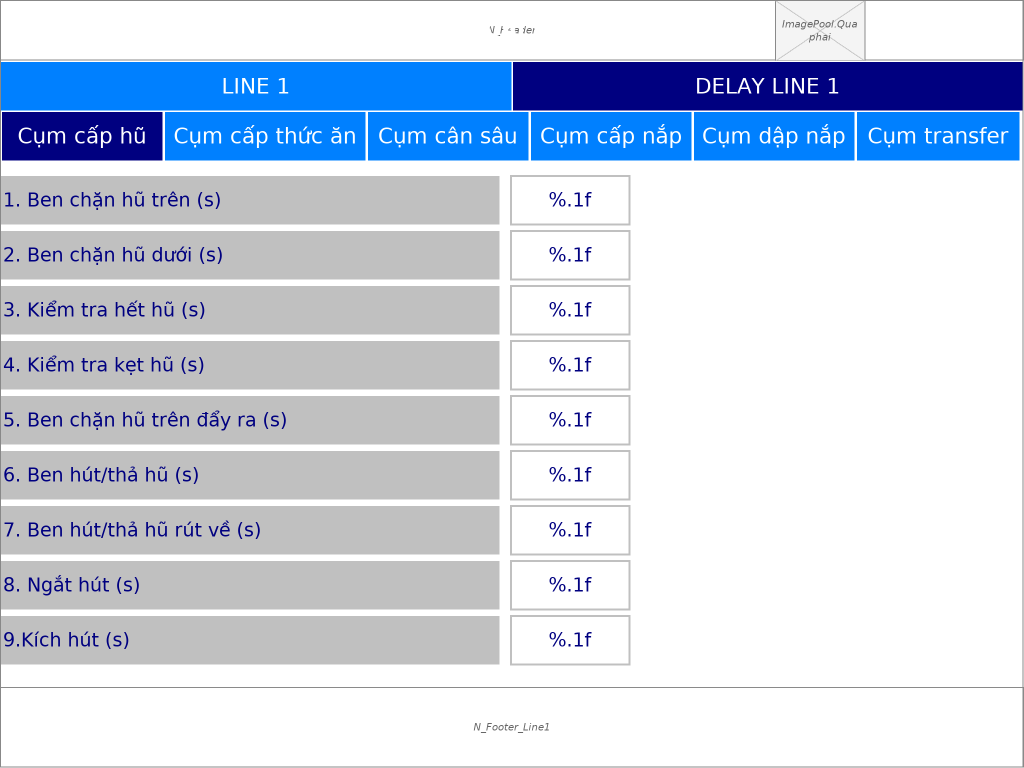
VISUALIZATION N_Setting_Delay_JarSupply1  // 1024x768
    Frame (0,687 1024x80)
        shows N_Footer_Line1()
    Frame (0,0 1024x60)
        shows N_Header()
    Textfield (353,4 420x50), "MÀN HÌNH CÀI KHOẢNG TRỄ LINE 1"
    Rectangle (0,61 512x50), "LINE 1"
        OnMouseClick: change screen: N_Setting_Line1
    Image (775,0 90x61), image: ImagePool.Qua phai
        OnMouseClick: change screen: N_Setting_Delay_JarSupply2
    Rectangle (1,111 162x50), "Cụm cấp hũ"
        OnMouseClick: change screen: N_Setting_Delay_JarSupply1
    Rectangle (164,111 202x50), "Cụm cấp thức ăn"
        OnMouseClick: change screen: N_Setting_Delay_FoodSupply1
    Rectangle (367,111 162x50), "Cụm cân sâu"
        OnMouseClick: change screen: N_Setting_Delay_WormWeight1
    Rectangle (530,111 162x50), "Cụm cấp nắp"
        OnMouseClick: change screen: N_Setting_Delay_LidSupply1
    Rectangle (693,111 162x50), "Cụm dập nắp"
        OnMouseClick: change screen: N_Setting_Delay_LidPressing1
    Rectangle (856,111 164x50), "Cụm transfer"
        OnMouseClick: change screen: N_Setting_Delay_Tranfer1
    Rectangle (512,61 511x50), "DELAY LINE 1"
        OnMouseClick: change screen: N_Setting_Delay_JarSupply1
    Rectangle (0,175 500x50), "1. Ben chặn hũ trên (s)"
    Rectangle (510,175 120x50), "%.1f", text variable: PR_Line01.timerCheckCylinder_Up
        OnMouseClick: write PR_Line01.timerCheckCylinder_Up via VisuDialogs.Numpad
    Rectangle (0,230 500x50), "2. Ben chặn hũ dưới (s)"
    Rectangle (510,230 120x50), "%.1f", text variable: PR_Line01.timerCheckCylinder_Dw
        OnMouseClick: write PR_Line01.timerCheckCylinder_Dw via VisuDialogs.Numpad
    Rectangle (0,340 500x50), "4. Kiểm tra kẹt hũ (s)"
    Rectangle (0,285 500x50), "3. Kiểm tra hết hũ (s)"
    Rectangle (510,285 120x50), "%.1f", text variable: PR_Line01.timerCheckEmpty
        OnMouseClick: write PR_Line01.timerCheckEmpty via VisuDialogs.Numpad
    Rectangle (510,340 120x50), "%.1f", text variable: PR_Line01.timerCheckStuck
        OnMouseClick: write PR_Line01.timerCheckStuck via VisuDialogs.Numpad
    Rectangle (0,395 500x50), "5. Ben chặn hũ trên đẩy ra (s)"
    Rectangle (510,395 120x50), "%.1f", text variable: PR_Line01.timerCylinder_Up_extend
        OnMouseClick: write PR_Line01.timerCylinder_Up_extend via VisuDialogs.Numpad
    Rectangle (0,450 500x50), "6. Ben hút/thả hũ (s)"
    Rectangle (510,450 120x50), "%.1f", text variable: PR_Line01.timerCylinder_Suction_Cup
        OnMouseClick: write PR_Line01.timerCylinder_Suction_Cup via VisuDialogs.Numpad
    Rectangle (0,505 500x50), "7. Ben hút/thả hũ rút về (s)"
    Rectangle (510,505 120x50), "%.1f", text variable: PR_Line01.timerCylinder_Suction_Cup_extend
        OnMouseClick: write PR_Line01.timerCylinder_Suction_Cup_extend via VisuDialogs.Numpad
    Rectangle (0,560 500x50), "8. Ngắt hút (s)"
    Rectangle (510,560 120x50), "%.1f", text variable: PR_Line01.timerCylinder_Suction_Val
        OnMouseClick: write PR_Line01.timerCylinder_Suction_Val via VisuDialogs.Numpad
    Rectangle (0,615 500x50), "9.Kích hút (s)"
    Rectangle (510,615 120x50), "%.1f", text variable: PR_Line01.timerCylinder_Suction_pick
        OnMouseClick: write PR_Line01.timerCylinder_Suction_pick via VisuDialogs.Numpad
END_VISUALIZATION

(* stored: Version 1.1.0.1, ProductVersion 3.1.4024.12
   Visu N_Setting_Delay_JarSupply1: Id {68023a8c-a24d-492a-821d-0f93ad0ca565} *)
